  990 = 'Mc_Prompts Default 990' | German: 'Mc_Prompts German 990' | French: 'Mc_Prompts French 990'
  991 = 'Mc_Prompts Default 991' | German: 'Mc_Prompts German 991' | French: 'Mc_Prompts French 991'
  992 = 'Mc_Prompts Default 992' | German: 'Mc_Prompts German 992' | French: 'Mc_Prompts French 992'
  993 = 'Mc_Prompts Default 993' | German: 'Mc_Prompts German 993' | French: 'Mc_Prompts French 993'
  994 = 'Mc_Prompts Default 994' | German: 'Mc_Prompts German 994' | French: 'Mc_Prompts French 994'
  995 = 'Mc_Prompts Default 995' | German: 'Mc_Prompts German 995' | French: 'Mc_Prompts French 995'
  996 = 'Mc_Prompts Default 996' | German: 'Mc_Prompts German 996' | French: 'Mc_Prompts French 996'
  997 = 'Mc_Prompts Default 997' | German: 'Mc_Prompts German 997' | French: 'Mc_Prompts French 997'
  998 = 'Mc_Prompts Default 998' | German: 'Mc_Prompts German 998' | French: 'Mc_Prompts French 998'
  999 = 'Mc_Prompts Default 999' | German: 'Mc_Prompts German 999' | French: 'Mc_Prompts French 999'
  1000 = 'Mc_Prompts Default 1000' | German: 'Mc_Prompts German 1000' | French: 'Mc_Prompts French 1000'
   = ''
END_TEXTLIST

(* stored: Version 1.1.0.1, ProductVersion 3.1.4024.11
   TextList Mc_Prompts: Id {503447e5-717e-0dc4-20dd-dba12d898279} *)
